INTERFACE I_GraphAddedEvent EXTENDS I_Event

PROPERTY PUBLIC Target : I_Graph
GET
END_GET
END_PROPERTY

END_INTERFACE

(* stored: Version 1.1.0.1, ProductVersion 3.1.4024.12
   Itf I_GraphAddedEvent: Id {c6433338-b296-4475-933e-3ef65a5a4bf7}
   Property Target: Id {f84e34f4-2ba9-444e-bc13-ef9d2a1b9a55}
   Get Get: Id {4854e24c-11f0-4a4a-ae94-5457e82fb0bb} *)
